                TPErase;
                TPWrite "Robot Axis 1 : "+ValToStr(rEmptyJoint.robax.rax_1)+"Robot Axis 2 : "+ValToStr(rEmptyJoint.robax.rax_2);
                TPWrite "Robot Axis 3 : "+ValToStr(rEmptyJoint.robax.rax_3)+"Robot Axis 4 : "+ValToStr(rEmptyJoint.robax.rax_4);
                TPWrite "Robot Axis 5 : "+ValToStr(rEmptyJoint.robax.rax_5)+"Robot Axis 6 : "+ValToStr(rEmptyJoint.robax.rax_6);

                TPReadFK n,"Right?","Yes",stEmpty,stEmpty,stEmpty,"No";
                IF n=5 GOTO gHomeStart;
                IF n=1 THEN
                    TPReadFK n,"Did you want Save Home Position?","Yes",stEmpty,stEmpty,stEmpty,"No";
                    IF n=5 GOTO gHomeStart;
                    TPErase;
                    TPWrite "Save Home Position";
                    jHomeJoint:=rEmptyJoint;
                    WaitTime 0.3;
                ENDIF
                GOTO gHomeStart;

            ELSEIF n=4 THEN
                TPWrite "Go Home Position";
                rMoveHome;
                !MoveAbsJ jHomeJoint, v300, fine, tool0;
                TPWrite "Arrived Homoe Position Go to Menu";
            ELSE

                TPWrite "Go To Menu";
                WaitTime 0.3;
                GOTO gStart;

            ENDIF

        CASE 5:
            TPWrite "Go To Menu";
            WaitTime 0.3;
            GOTO gStart;
        ENDTEST

        gAuto:

    ENDPROC

    PROC rWirecut(num nRbt_No)
        bWirecut:=[FALSE,FALSE,FALSE];
        IF (sdo_Rob_1_JgHome=1 AND sdo_Rob_2_JgHome=1) OR (sdo_Rob_1_MoveHome=1 AND sdo_Rob_2_MoveHome=1) OR (sdo_Rob_1_WirecutHome=1 AND sdo_Rob_2_WirecutHome=1) THEN
        ELSE
            rMeasurementHomeCheck;
        ENDIF
        IF sdo_Rob_1_JgHome=1 AND sdo_Rob_2_JgHome=1 THEN
            bWirecut:=[TRUE,FALSE,FALSE];
            IF nRbt_No=0 OR nRbt_No=1 THEN
                Wirecut\R1;
                WaitUntil stReact{1}="WireCutOk";
                stCommand:="";
                WaitUntil stReact{1}="Ready";
            ENDIF
            IF nRbt_No=0 OR nRbt_No=2 THEN
                WireCut\R2;
                WaitUntil stReact{2}="WireCutOk";
                stCommand:="";
                WaitUntil stReact{2}="Ready";
            ENDIF
            IF nRbt_No=3 THEN
                bWireCutSync:=TRUE;
                stCommand:="WireCutR1_R2";
                WaitUntil stReact{1}="WireCutOk" AND stReact{2}="WireCutOk";
                stCommand:="";
                WaitUntil stReact{1}="Ready" AND stReact{2}="Ready";
                bWireCutSync:=FALSE;
            ENDIF
        ENDIF
        IF sdo_Rob_1_MoveHome=1 AND sdo_Rob_2_MoveHome=1 THEN
            bWirecut:=[FALSE,TRUE,FALSE];
            IF nRbt_No=0 OR nRbt_No=1 THEN
                WirecutMove\R1;
                WaitUntil stReact{1}="WireCutOk";
                stCommand:="";
                WaitUntil stReact{1}="Ready";
            ENDIF
            IF nRbt_No=0 OR nRbt_No=2 THEN
                WireCutMove\R2;
                WaitUntil stReact{2}="WireCutOk";
                stCommand:="";
                WaitUntil stReact{2}="Ready";
            ENDIF
            IF nRbt_No=3 THEN
                bWireCutSync:=TRUE;
                stCommand:="WireCutMoveR1_R2";
                WaitUntil stReact{1}="WireCutOk" AND stReact{2}="WireCutOk";
                stCommand:="";
                WaitUntil stReact{1}="Ready" AND stReact{2}="Ready";
                bWireCutSync:=FALSE;
            ENDIF
        ENDIF
        IF sdo_Rob_1_WirecutHome=1 AND sdo_Rob_2_WirecutHome=1 THEN
            bWirecut:=[FALSE,FALSE,TRUE];
            IF nRbt_No=0 OR nRbt_No=1 THEN
                WirecutShot\R1;
                WaitUntil stReact{1}="WireCutOk";
                stCommand:="";
                WaitUntil stReact{1}="Ready";
            ENDIF
            IF nRbt_No=0 OR nRbt_No=2 THEN
                WireCutShot\R2;
                WaitUntil stReact{2}="WireCutOk";
                stCommand:="";
                WaitUntil stReact{2}="Ready";
            ENDIF
            IF nRbt_No=3 THEN
                bWireCutSync:=TRUE;
                stCommand:="WireCutShotR1_R2";
                WaitUntil stReact{1}="WireCutOk" AND stReact{2}="WireCutOk";
                stCommand:="";
                WaitUntil stReact{1}="Ready" AND stReact{2}="Ready";
                bWireCutSync:=FALSE;
            ENDIF
        ENDIF
        WaitUntil stReact=["Ready","Ready","Ready"];

    ENDPROC

    PROC rWirecutShot(num nRbt_No)

        IF nRbt_No=0 OR nRbt_No=1 THEN
            WirecutShot\R1;
            WaitUntil stReact{1}="WireCutOk";
            stCommand:="";
            WaitUntil stReact{1}="Ready";
        ENDIF
        IF nRbt_No=0 OR nRbt_No=2 THEN
            WireCutShot\R2;
            WaitUntil stReact{2}="WireCutOk";
            stCommand:="";
            WaitUntil stReact{2}="Ready";
        ENDIF
        IF nRbt_No=3 THEN
            bWireCutSync:=TRUE;
            stCommand:="WireCutShotR1_R2";
            WaitUntil stReact{1}="WireCutOk" AND stReact{2}="WireCutOk";
            stCommand:="";
            WaitUntil stReact{1}="Ready" AND stReact{2}="Ready";
            bWireCutSync:=FALSE;
        ENDIF

        WaitUntil stReact=["Ready","Ready","Ready"];

    ENDPROC

    PROC rWirecutMove(num nRbt_No)

        IF nRbt_No=0 OR nRbt_No=1 THEN
            WirecutMove\R1;
            WaitUntil stReact{1}="WireCutOk";
            stCommand:="";
            WaitUntil stReact{1}="Ready";
        ENDIF
        IF nRbt_No=0 OR nRbt_No=2 THEN
            WireCutMove\R2;
            WaitUntil stReact{2}="WireCutOk";
            stCommand:="";
            WaitUntil stReact{2}="Ready";
        ENDIF
        IF nRbt_No=3 THEN
            bWireCutSync:=TRUE;
            stCommand:="WireCutMoveR1_R2";
            WaitUntil stReact{1}="WireCutOk" AND stReact{2}="WireCutOk";
            stCommand:="";
            WaitUntil stReact{1}="Ready" AND stReact{2}="Ready";
            bWireCutSync:=FALSE;
        ENDIF

        WaitUntil stReact=["Ready","Ready","Ready"];

    ENDPROC

    PROC rEdgeDataCheck()
        IF edgeStart{1}.Breadth<=0 edgeStart{1}.Breadth:=50;
        IF edgeStart{1}.Height<=0 edgeStart{1}.Height:=50;
        IF edgeStart{2}.Breadth<=0 edgeStart{2}.Breadth:=50;
        IF edgeStart{2}.Height<=0 edgeStart{2}.Height:=50;
        IF edgeEnd{1}.Breadth<=0 edgeEnd{1}.Breadth:=50;
        IF edgeEnd{1}.Height<=0 edgeEnd{1}.Height:=50;
        IF edgeEnd{2}.Breadth<=0 edgeEnd{2}.Breadth:=50;
        IF edgeEnd{2}.Height<=0 edgeEnd{2}.Height:=50;
    ENDPROC

    PROC rMoveHome_Head()

        WaitUntil stReact=["Error_Arc_Touch","Error_Arc_Touch","Error_Arc_Touch"];
        stCommand:="Error_Arc_Touch";
        WaitUntil stReact=["","",""];
        stCommand:="";
        WaitUntil stReact=["","",""];
        nErrorCmd:=1;
        ExitCycle;

    ENDPROC

    PROC rWireReplacementMode()
        VAR jointgroup jTempReadyGroup;
        VAR num nTempChangPos;
        VAR num nMaxHeight;
        !!!!!!==MoveToHome==,[
        rMeasurementHomeCheck;

        jTempReadyGroup:=MergeJgWith();
        jTempReadyGroup.JointG.extax.eax_b:=Limit(0,5300,nLimitY_Positive-nMaintenanceYPos);
        MoveJgJ MergeJgWith(\Gantry:=jTempReadyGroup.JointG),vTargetSpeed,z200;

        jTempReadyGroup.JointG.extax.eax_c:=700;
        MoveJgJ MergeJgWith(\Gantry:=jTempReadyGroup.JointG),vTargetSpeed,z200;

        RETURN ;
    ENDPROC

    PROC rArcErrorGantryDown()
        VAR jointgroup jTempReadyGroup;
        VAR num nTempGantryHeight;
        VAR num nTempPartHeightTemp;
        jTempReadyGroup:=MergeJgWith();
        nTempPartHeightTemp:=max(max(nMaxPartHeightNearArray{1},nMaxPartHeightNearArray{2}),nMaxPartHeightNearArray{3});

        nTempGantryHeight:=nHomeGantryZ-(900+nTempPartHeightTemp);
        jTempReadyGroup.JointG.extax.eax_c:=nTempGantryHeight;
        jTempReadyGroup.JointG.extax.eax_c:=Limit(0,1000,jTempReadyGroup.JointG.extax.eax_c);
        MoveJgJ MergeJgWith(\Gantry:=jTempReadyGroup.JointG),vTargetSpeed,z200;
    ENDPROC

    PROC rMeasurementHomeCheck()
        VAR jointgroup jMeasurementHomeGroup;
        VAR bool bHomeCheck:=FALSE;
        bHomeCheck:=FALSE;
        jMeasurementHomeGroup:=MergeJgWith();
        IF abs(jMeasurementHomeGroup.Joint1.robax.rax_1-jgMeasurementHome.Joint1.robax.rax_1)>1 bHomeCheck:=TRUE;
        IF abs(jMeasurementHomeGroup.Joint1.robax.rax_2-jgMeasurementHome.Joint1.robax.rax_2)>1 bHomeCheck:=TRUE;
        IF abs(jMeasurementHomeGroup.Joint1.robax.rax_3-jgMeasurementHome.Joint1.robax.rax_3)>1 bHomeCheck:=TRUE;
        IF abs(jMeasurementHomeGroup.Joint1.robax.rax_4-jgMeasurementHome.Joint1.robax.rax_4)>1 bHomeCheck:=TRUE;
        IF abs(jMeasurementHomeGroup.Joint1.robax.rax_5-jgMeasurementHome.Joint1.robax.rax_5)>1 bHomeCheck:=TRUE;
        IF abs(jMeasurementHomeGroup.Joint1.robax.rax_6-jgMeasurementHome.Joint1.robax.rax_6)>1 bHomeCheck:=TRUE;
        IF abs(jMeasurementHomeGroup.Joint2.robax.rax_1-jgMeasurementHome.Joint2.robax.rax_1)>1 bHomeCheck:=TRUE;
        IF abs(jMeasurementHomeGroup.Joint2.robax.rax_2-jgMeasurementHome.Joint2.robax.rax_2)>1 bHomeCheck:=TRUE;
        IF abs(jMeasurementHomeGroup.Joint2.robax.rax_3-jgMeasurementHome.Joint2.robax.rax_3)>1 bHomeCheck:=TRUE;
        IF abs(jMeasurementHomeGroup.Joint2.robax.rax_4-jgMeasurementHome.Joint2.robax.rax_4)>1 bHomeCheck:=TRUE;
        IF abs(jMeasurementHomeGroup.Joint2.robax.rax_5-jgMeasurementHome.Joint2.robax.rax_5)>1 bHomeCheck:=TRUE;
        IF abs(jMeasurementHomeGroup.Joint2.robax.rax_6-jgMeasurementHome.Joint2.robax.rax_6)>1 bHomeCheck:=TRUE;

        IF bHomeCheck=TRUE THEN
            rByTaskMoveToRobotHome 1;
        ELSE
            jMeasurementHomeGroup.JointG.extax.eax_c:=0;
            MoveJgJ jMeasurementHomeGroup,vTargetSpeed,fine;
        ENDIF
    ENDPROC

    PROC rjgWireCutHomeCheck()
        VAR jointgroup jWirecutHomeGroup;
        VAR bool bHomeCheck:=FALSE;
        bHomeCheck:=FALSE;
        jWirecutHomeGroup:=MergeJgWith();

        IF abs(jWirecutHomeGroup.Joint1.robax.rax_1-jgWireCutHome.Joint1.robax.rax_1)>1 bHomeCheck:=TRUE;
        IF abs(jWirecutHomeGroup.Joint1.robax.rax_2-jgWireCutHome.Joint1.robax.rax_2)>1 bHomeCheck:=TRUE;
        IF abs(jWirecutHomeGroup.Joint1.robax.rax_3-jgWireCutHome.Joint1.robax.rax_3)>1 bHomeCheck:=TRUE;
        IF abs(jWirecutHomeGroup.Joint1.robax.rax_4-jgWireCutHome.Joint1.robax.rax_4)>1 bHomeCheck:=TRUE;
        IF abs(jWirecutHomeGroup.Joint1.robax.rax_5-jgWireCutHome.Joint1.robax.rax_5)>1 bHomeCheck:=TRUE;
        IF abs(jWirecutHomeGroup.Joint1.robax.rax_6-jgWireCutHome.Joint1.robax.rax_6)>1 bHomeCheck:=TRUE;
        IF abs(jWirecutHomeGroup.Joint2.robax.rax_1-jgWireCutHome.Joint2.robax.rax_1)>1 bHomeCheck:=TRUE;
        IF abs(jWirecutHomeGroup.Joint2.robax.rax_2-jgWireCutHome.Joint2.robax.rax_2)>1 bHomeCheck:=TRUE;
        IF abs(jWirecutHomeGroup.Joint2.robax.rax_3-jgWireCutHome.Joint2.robax.rax_3)>1 bHomeCheck:=TRUE;
        IF abs(jWirecutHomeGroup.Joint2.robax.rax_4-jgWireCutHome.Joint2.robax.rax_4)>1 bHomeCheck:=TRUE;
        IF abs(jWirecutHomeGroup.Joint2.robax.rax_5-jgWireCutHome.Joint2.robax.rax_5)>1 bHomeCheck:=TRUE;
        IF abs(jWirecutHomeGroup.Joint2.robax.rax_6-jgWireCutHome.Joint2.robax.rax_6)>1 bHomeCheck:=TRUE;

        IF bHomeCheck=TRUE THEN
            rByTaskMoveToRobotHome 2;
        ELSE
            jWirecutHomeGroup.JointG.extax.eax_c:=0;
            MoveJgJ jWirecutHomeGroup,vTargetSpeed,fine;
        ENDIF
    ENDPROC

    PROC rByTaskMoveToRobotHome(num nHomeNo)
        VAR jointgroup jgEmptyTarget;
        VAR jointtarget jTempG;
        VAR num ntemp;

        stCommand:="checkpos";
        waituntil stReact=["checkposok","checkposok","checkposok"];
        stCommand:="";
        waituntil stReact=["Ready","Ready","Ready"];

        jgEmptyTarget.Joint1:=CJointT(\TaskName:="T_Rob1");
        jgEmptyTarget.Joint2:=CJointT(\TaskName:="T_Rob2");
        jgEmptyTarget.JointG:=CJointT(\TaskName:="T_Gantry");
        jgEmptyTarget.JointG.extax.eax_c:=0;
        MoveJgJ jgEmptyTarget,vTargetSpeed,fine;

        jgEmptyTarget.Joint1.robax.rax_2:=-90;
        jgEmptyTarget.Joint1.robax.rax_3:=55;
        jgEmptyTarget.Joint2.robax.rax_2:=-90;
        jgEmptyTarget.Joint2.robax.rax_3:=55;
        MoveJgJ jgEmptyTarget,vTargetSpeed,fine;

        jgEmptyTarget.Joint1.robax.rax_5:=0;
        jgEmptyTarget.Joint2.robax.rax_5:=0;
        MoveJgJ jgEmptyTarget,vTargetSpeed,fine;
        IF nHomeNo=1 THEN
            jgEmptyTarget.Joint1.robax.rax_1:=jgMeasurementHome.Joint1.robax.rax_1;
            jgEmptyTarget.Joint2.robax.rax_1:=jgMeasurementHome.Joint2.robax.rax_1;
        ELSEIF nHomeNo=2 THEN
            jgEmptyTarget.Joint1.robax.rax_1:=jgWireCutHome.Joint1.robax.rax_1;
            jgEmptyTarget.Joint2.robax.rax_1:=jgWireCutHome.Joint2.robax.rax_1;
        ENDIF
        jgEmptyTarget.JointG.extax.eax_d:=0;
        MoveJgJ jgEmptyTarget,vTargetSpeed,fine;

        jgEmptyTarget.Joint1:=CJointT(\TaskName:="T_Rob1");
        jgEmptyTarget.Joint2:=CJointT(\TaskName:="T_Rob2");
        jgEmptyTarget.JointG:=CJointT(\TaskName:="T_Gantry");
        IF nHomeNo=1 THEN
            jgEmptyTarget.Joint1.robax:=jgMeasurementHome.Joint1.robax;
            jgEmptyTarget.Joint2.robax:=jgMeasurementHome.Joint2.robax;
        ELSEIF nHomeNo=2 THEN
            jgEmptyTarget.Joint1.robax:=jgWireCutHome.Joint1.robax;
            jgEmptyTarget.Joint2.robax:=jgWireCutHome.Joint2.robax;
        ENDIF
        MoveJgJ jgEmptyTarget,vTargetSpeed,fine;

        RETURN ;
    ENDPROC

   PROC rWarm_Up()

        VAR speeddata vWarmUp_Speed;
        VAR num i:=0;
        VAR num nWarmUp_Distance_X;
        VAR num nWarmUp_Distance_Y;
        VAR num nWarmUp_Distance_Z;
        VAR num nWarmUp_Distance_R;
        VAR num nTempDistance:=0;
        VAR clock clWarmUp;
        VAR bool bWarmUpComplete:=FALSE;
        VAR jointgroup jgWarmUpTargetpos;
        VAR num nWarmUp_Target_X:=0;


        !..... Userset Gantry_X .........
        nWarmUp_Target_X:=12000;
        !................................
        jgWarmUpTargetpos:=jgHomeJoint;
        jgWarmUpTargetpos.JointG.extax.eax_a:=nWarmUp_Target_X;
        jgWarmUpTargetpos.JointG.extax.eax_f:=nWarmUp_Target_X;

        jgTarget:=MergeJgWith();
        jgTarget.JointG:=jgWarmUpTargetpos.JointG;
        jgTarget.JointG.extax.eax_d:=90;

        vWarmUp_Speed:=[300,300,10,10];
        ClkReset clWarmUp;
        ClkStart clWarmUp;

        WHILE bWarmUpComplete=FALSE DO

            jgWarm_Up:=MergeJgWith();

            ! eax_a
            IF jgWarm_Up.JointG.extax.eax_a<jgWarmUpTargetpos.JointG.extax.eax_a+149 AND jgWarm_Up.JointG.extax.eax_a>jgWarmUpTargetpos.JointG.extax.eax_a-149 THEN
                jgTarget.JointG.extax.eax_a:=jgWarmUpTargetpos.JointG.extax.eax_a-150;
            ELSE
                IF jgWarm_Up.JointG.extax.eax_a<jgWarmUpTargetpos.JointG.extax.eax_a-150 jgTarget.JointG.extax.eax_a:=jgWarmUpTargetpos.JointG.extax.eax_a+150;
            ENDIF
            nWarmUp_Distance_X:=jgTarget.JointG.extax.eax_a-jgWarm_Up.JointG.extax.eax_a;
            IF nWarmUp_Distance_X>0 THEN
                nTempDistance:=100;
            ELSE
                nTempDistance:=-100;
            ENDIF
            jgWarm_Up.JointG.extax.eax_a:=jgWarm_Up.JointG.extax.eax_a+nTempDistance;
            jgWarm_Up.JointG.extax.eax_f:=jgWarm_Up.JointG.extax.eax_f+nTempDistance;

            ! eax_b
            IF jgWarm_Up.JointG.extax.eax_b>149 jgTarget.JointG.extax.eax_b:=0;
            IF jgWarm_Up.JointG.extax.eax_b<1 jgTarget.JointG.extax.eax_b:=150;
            nWarmUp_Distance_Y:=jgTarget.JointG.extax.eax_b-jgWarm_Up.JointG.extax.eax_b;
            IF nWarmUp_Distance_Y>0 THEN
                nTempDistance:=100;
            ELSE
                nTempDistance:=-100;
            ENDIF
            jgWarm_Up.JointG.extax.eax_b:=jgWarm_Up.JointG.extax.eax_b+nTempDistance;

            ! eax_c
            IF jgWarm_Up.JointG.extax.eax_c<1 jgTarget.JointG.extax.eax_c:=100;
            IF jgWarm_Up.JointG.extax.eax_c>99 jgTarget.JointG.extax.eax_c:=0;
            nWarmUp_Distance_Z:=jgTarget.JointG.extax.eax_c-jgWarm_Up.JointG.extax.eax_c;
            IF nWarmUp_Distance_Z>0 THEN
                nTempDistance:=100;
            ELSE
                nTempDistance:=-100;
            ENDIF
            jgWarm_Up.JointG.extax.eax_c:=jgWarm_Up.JointG.extax.eax_c+nTempDistance;

            ! eax_d
            IF jgWarm_Up.JointG.extax.eax_d<-81 jgTarget.JointG.extax.eax_d:=90;
            IF jgWarm_Up.JointG.extax.eax_d>81 jgTarget.JointG.extax.eax_d:=-90;
            nWarmUp_Distance_R:=jgTarget.JointG.extax.eax_d-jgWarm_Up.JointG.extax.eax_d;
            IF nWarmUp_Distance_R>0 THEN
                nTempDistance:=10;
            ELSE
                nTempDistance:=-10;
            ENDIF
            jgWarm_Up.JointG.extax.eax_d:=jgWarm_Up.JointG.extax.eax_d+nTempDistance;

            !  move
            jgWarm_Up.JointG.extax.eax_b:=Limit(0,5300,jgWarm_Up.JointG.extax.eax_b);
            jgWarm_Up.JointG.extax.eax_c:=Limit(0,100,jgWarm_Up.JointG.extax.eax_c);
            jgWarm_Up.JointG.extax.eax_d:=Limit(-90,90,jgWarm_Up.JointG.extax.eax_d);
            MoveJgJ MergeJgWith(\Gantry:=jgWarm_Up.JointG),vWarmUp_Speed,fine;
            vWarmUp_Speed.v_reax:=vWarmUp_Speed.v_reax+0.1;
            vWarmUp_Speed.v_leax:=vWarmUp_Speed.v_leax+0.5;
            IF vWarmUp_Speed.v_reax>25 vWarmUp_Speed.v_reax:=25;
            IF vWarmUp_Speed.v_leax>250 vWarmUp_Speed.v_leax:=250;
            nWarmUpTime:=ClkRead(clWarmUp);
            IF nWarmUpTime>nWarmUpCycle bWarmUpComplete:=TRUE;
        ENDWHILE
        ClkStop clWarmUp;
        RETURN ;
    ENDPROC

    PROC rGantry_C_Home()
        VAR jointgroup jgGantry_C_Home;
        jgGantry_C_Home:=MergeJgWith();
        jgGantry_C_Home.JointG.extax.eax_c:=0;
        MoveJgJ MergeJgWith(\Gantry:=jgGantry_C_Home.JointG),vTargetSpeed,fine;
        WaitRob\InPos;
        WaitRob\ZeroSpeed;
    ENDPROC
ENDMODULE
